PROGRAM MAIN
VAR_INPUT
	// open the roof remotely
	OpenRoofAuto: 	BOOL;
	// close the roof remotely
	CloseRoofAuto: 	BOOL;
	// stop the roof remotely (unused?)
	StopRoofAuto: 	BOOL;
	// turn on the light remotely
	LightAuto: 		BOOL;
END_VAR

VAR
	// RoofManual or RoofAutomatic
	nMode:		    E_RoofMode;
	// DachControl roof1
	Dach1Control:	FB_RoofControl;
	// DachControl roof 2
	Dach2Control:	FB_RoofControl;
	Roof1Command,
	Roof2Command:	E_RoofCommand;
	Roof1Status,
	Roof2Status,
	LastRoof1Status,
	LastRoof2Status:	E_RoofStatus;
	RSOpenRoof1,
	RSCloseRoof1,
	RSOpenRoof2,
	RSCloseRoof2: 	RS;
	OpenRoofAutoPending: BOOL;
	OpenRoof1,
	CloseRoof1,
	OpenRoof2,
	CloseRoof2,
	StopRoof1,
	StopRoof2:	BOOL;
	// report manual operation of the dome to TCS
	isRoofManual: BOOL;
	// indicates an error in the dust sensor
	DustSensorError: BOOL;
	// Timer for Dome Light
	LightTimer:		LIGHT_BUTTON;

	RoofStatusLamp1,
	RoofStatusLamp2: FB_StatusLamp;
	WeatherAlarm,
	MotionAlarm1,
	MotionAlarm2:	BOOL;
	// indicates at least on environment signal is bad
	EnvironmentBad,
	// environment signal is bad for n seconds
	EnvironmentAlarm: BOOL;
	// time function block for Environment signal
	EnvironmentBadTimer: TON;
	MQTTTimer : TON := (PT:=T#5S);
	// MQTT class for publishing
	MQTTClient:		FB_MQTTCommunication;
	// Humidity Trigger
	HumidityTrigger:	SR;
	Roof1OpenTimer,
	Roof2OpenTimer,
	Roof1CloseTimer,
	Roof2CloseTimer:	TIMER;
	Roof1OpenTimeOut,
	Roof2OpenTimeOut,
	Roof1CloseTimeOut,
	Roof2CloseTimeOut:	TON;
END_VAR
VAR CONSTANT
	HumidityLimitHigh:		REAL := 80.0;
	HumidityLimitLow:		REAL := 65.0;
	
	WindSpeedLimit:		REAL := 20.0;
	WindSpeedBayLimit:	REAL :=	15.0;
	DustLimit:			REAL := 0.01;
	BrightnessLimit:	REAL := 40000.0;
END_VAR

IF GVL_Panel.IManualSwitch THEN
	nMode := RoofManual;
ELSE
	nMode := RoofAutomatic;
END_IF
isRoofManual := GVL_Panel.IManualSwitch;

DustSensorError := GVL_Environment.DustSensorError;

// initialize MQTT Communication
MQTTClient();

// collect weather data
Environment();

// Handle Auxiliary inputs and outputs
Auxiliary();

// Handle Logging
Logging();

// Control Logic for Dehumidifier
DehumidifierControl(Enable := nMode = RoofAutomatic AND Roof1Status = StatusLocked AND Roof2Status = StatusLocked);

HumidityTrigger(SET1 := Environment.Humidity >= HumidityLimitHigh,
				RESET := Environment.Humidity < HumidityLimitLow);
						
// define bad weather condition; rain is handled in EnvironmentAlarm
EnvironmentBad := (Environment.Dust > DustLimit AND NOT DustSensorError) OR
		HumidityTrigger.Q1 OR
		Environment.WindSpeed1 > WindSpeedLimit OR
		Environment.WindSpeed2 > WindSpeedLimit OR
		Environment.Windspeed_bay > WindSpeedBayLimit; // OR
		//ConvertEnvironment.Brightness > BrightnessLimit;

EnvironmentBadTimer(IN := EnvironmentBad,
					PT := T#125S);
					
EnvironmentAlarm := EnvironmentBadTimer.Q OR Environment.RainMasterAlarm;

IF nMode = RoofAutomatic THEN
	// if we get the open comand during bad weather, postpone the signal
	IF OpenRoofAuto AND EnvironmentAlarm THEN
		OpenRoofAutoPending := TRUE;
		OpenRoofAuto := FALSE;
	// if we get the close command cancle the signal
	ELSIF CloseRoofAuto THEN
		OpenRoofAutoPending := FALSE;
	END_IF
	// if weather is good, execute the pending signal
	IF NOT EnvironmentAlarm AND OpenRoofAutoPending THEN
		OpenRoofAuto := TRUE;
		OpenRoofAutoPending := FALSE;
	END_IF			

	IF OpenRoofAuto THEN
		Roof1Command := OpenRoof;
		Roof2Command := OpenRoof;
	ELSIF CloseRoofAuto THEN
		Roof1Command := CloseRoof;
		Roof2Command := CloseRoof;
	ELSE
		Roof1Command := StopRoof;
		Roof2Command := StopRoof;
	END_IF

	// overwrite previous command if the weather is bad for xx seconds
	IF EnvironmentAlarm THEN
		IF NOT (Roof1Status = StatusLocked) THEN
			Roof1Command := CloseRoof;	
		END_IF
		IF NOT (Roof2Status = StatusLocked) THEN
			Roof2Command := CloseRoof;	
		END_IF
	END_IF
				
ELSE //	RoofManual
	OpenRoof1 := GVL_Panel.ILeftOpenSwitch AND NOT GVL_Panel.ILeftCloseSwitch;
	CloseRoof1 := GVL_Panel.ILeftCloseSwitch AND NOT GVL_Panel.ILeftOpenSwitch;
	StopRoof1 := NOT (GVL_Panel.ILeftOpenSwitch XOR GVL_Panel.ILeftCloseSwitch);
	
	IF OpenRoof1 THEN
		Roof1Command := OpenRoof;
	ELSIF CloseRoof1 THEN
		Roof1Command := CloseRoof;
	ELSE
		Roof1Command := StopRoof;
	END_IF

	OpenRoof2 := GVL_Panel.IRightOpenSwitch AND NOT GVL_Panel.IRightCloseSwitch;
	CloseRoof2 := GVL_Panel.IRightCloseSwitch AND NOT GVL_Panel.IRightOpenSwitch;
	StopRoof2 := NOT (GVL_Panel.IRightOpenSwitch XOR GVL_Panel.IRightCloseSwitch);
	
	IF OpenRoof2 THEN
		Roof2Command := OpenRoof;
	ELSIF CloseRoof2 THEN
		Roof2Command := CloseRoof;
	ELSE
		Roof2Command := StopRoof;
	END_IF
	Weatheralarm := ((Roof1Status = StatusOpened) OR (Roof2Status = StatusOpened))
					AND EnvironmentAlarm;
		
END_IF

Roof1OpenTimer(bStart := (Roof1Command = OpenRoof) AND NOT (Roof1Status = StatusOpened));
Roof2OpenTimer(bStart := (Roof2Command = OpenRoof) AND NOT (Roof2Status = StatusOpened));
Roof1CloseTimer(bStart := (Roof1Command = CloseRoof) AND NOT (Roof1Status = StatusLocked));
Roof2CloseTimer(bStart := (Roof2Command = CloseRoof) AND NOT (Roof2Status = StatusLocked));

Roof1OpenTimeOut(IN := (Roof1Command = OpenRoof) AND NOT (Roof1Status = StatusOpened), PT := T#130S);
Roof2OpenTimeOut(IN := (Roof2Command = OpenRoof) AND NOT (Roof2Status = StatusOpened), PT := T#130S);
Roof1CloseTimeOut(IN := (Roof1Command = CloseRoof) AND NOT (Roof1Status = StatusLocked), PT := T#130S);
Roof2CloseTimeOut(IN := (Roof1Command = CloseRoof) AND NOT (Roof2Status = StatusLocked), PT := T#130S);

	
// disable light after 1 hour if on automatic
LightTimer( IN := GVL_Environment.LightSwitch AND nMode = RoofAutomatic AND LightAuto,
			PT := T#1H);
			
GVL_Environment.LightBay := LightTimer.Q OR (nMode = RoofManual AND GVL_Environment.LightSwitch);	
// reset LightAuto SIgnal after one hour
IF nMode = RoofAutomatic AND LightAuto AND NOT LightTimer.Q1 THEN
	LightAuto := FALSE;
END_IF

(*** Control Section ***)	

Dach1Control(   cmdRoofCommand := Roof1Command,
				bOpenSwitch1   := GVL_Roof.IDach1auf,
				bOpenSwitch2   := GVL_Roof.IDach1auf2,
				bClosedSwitch1 := GVL_Roof.IDach1zu,
				bClosedSwitch2 := GVL_Roof.IDach1zu2,
				bLocked1       := GVL_Roof.IRiegel11zu,
				bUnlocked1     := GVL_Roof.IRiegel11auf,
				bLocked2       := GVL_Roof.IRiegel21zu,
				bUnlocked2     := GVL_Roof.IRiegel21auf,
				bFastSwitch    := GVL_Roof.IDach1Schnell,
				bOpenLock1     => GVL_Roof.ORiegel11auf,
				bCloseLock1    => GVL_Roof.ORiegel11zu,
				bOpenLock2     => GVL_Roof.ORiegel21auf,
				bCloseLock2    => GVL_Roof.ORiegel21zu,
				bRoofOpen 	   => GVL_Roof.ODach1auf,
				bRoofClose     => GVL_Roof.ODach1zu,
				bMotorFast     => GVL_Roof.ODach1Schnell,
				RoofStatus     => Roof1Status,
				MotionAlarm    => MotionAlarm1);

Dach2Control(   cmdRoofCommand := Roof2Command,
				bOpenSwitch1   := GVL_Roof.IDach2auf,
				bOpenSwitch2   := GVL_Roof.IDach2auf2,
				bClosedSwitch1 := GVL_Roof.IDach2zu,
				bClosedSwitch2 := GVL_Roof.IDach2zu2,
				bLocked1       := GVL_Roof.IRiegel12zu,
				bUnlocked1     := GVL_Roof.IRiegel12auf,
				bLocked2       := GVL_Roof.IRiegel22zu,
				bUnlocked2     := GVL_Roof.IRiegel22auf,
				bFastSwitch    := GVL_Roof.IDach2Schnell,
				bOpenLock1     => GVL_Roof.ORiegel12auf,
				bCloseLock1    => GVL_Roof.ORiegel12zu,
				bOpenLock2     => GVL_Roof.ORiegel22auf,
				bCloseLock2    => GVL_Roof.ORiegel22zu,
				bRoofOpen      => GVL_Roof.ODach2auf,
				bRoofClose     => GVL_Roof.ODach2zu,
				bMotorFast     => GVL_Roof.ODach2Schnell,
				RoofStatus     => Roof2Status,
				MotionAlarm    => MotionAlarm2);


// Set status lamps
RoofStatusLamp1(RoofStatus := Roof1Status, RoofLamp => GVL_Panel.Roof1Lamp);
RoofStatusLamp2(RoofStatus := Roof2Status, RoofLamp => GVL_Panel.Roof2Lamp);
			
// sound horn
GVL_Environment.Horn := WeatherAlarm OR MotionAlarm1 OR MotionAlarm2;		

IF GVL_Panel.Us_Undervoltage OR GVL_Panel.Up_Undervoltage THEN
	Roof1Status := StatusError;
	Roof2Status := StatusError;
END_IF


(*** MQTT Section ***)
MQTTTimer(IN:=TRUE);
IF MQTTTimer.Q OR Roof1Status <> LastRoof1Status OR Roof2Status <> LastRoof2Status THEN
	MQTTClient.Publish('roof', 'roof1', 'Roof1Status', RoofStatus_TO_String(Roof1Status));
	MQTTClient.Publish('roof', 'roof2', 'Roof2Status', RoofStatus_TO_String(Roof2Status));
	MAIN.MQTTClient.Publish('environment', 'weatherstation', 'WeatherBad',	BOOL_TO_STRING(EnvironmentAlarm));		
	MAIN.MQTTClient.Publish('roof', 'main', 'isRoofManual',	BOOL_TO_STRING(isRoofManual));		
	
	MQTTTimer(IN:=FALSE);
	LastRoof1Status := Roof1Status;
	LastRoof2Status := Roof2Status;
END_IF

END_PROGRAM

(* stored: Version 1.1.0.1, ProductVersion 3.1.4024.9
   POU MAIN: Id {a96e5090-a34b-4fcc-a0b3-91ecf58e0624}, SpecialFunc None *)
